TYPE ST_SensorData :
STRUCT
    rTemperature : REAL;
    rPressure    : REAL;
    bAlarm       : BOOL;
END_STRUCT
END_TYPE

(* stored: Version 1.1.0.1, ProductVersion 3.1.4024.16
   DUT ST_SensorData: Id {c4d19df8-32b6-4b09-b24f-edeea1c3c52a} *)
